// LS Electric XG5000 project: 과년68_3_3
// PLC NewPLC
// module base 0 slot 0: 입출력 모듈:XBC-DR20S (DC 24V 입력 12점, 릴레이 출력 8점)

PROGRAM NewProgram (task: 스캔 프로그램)

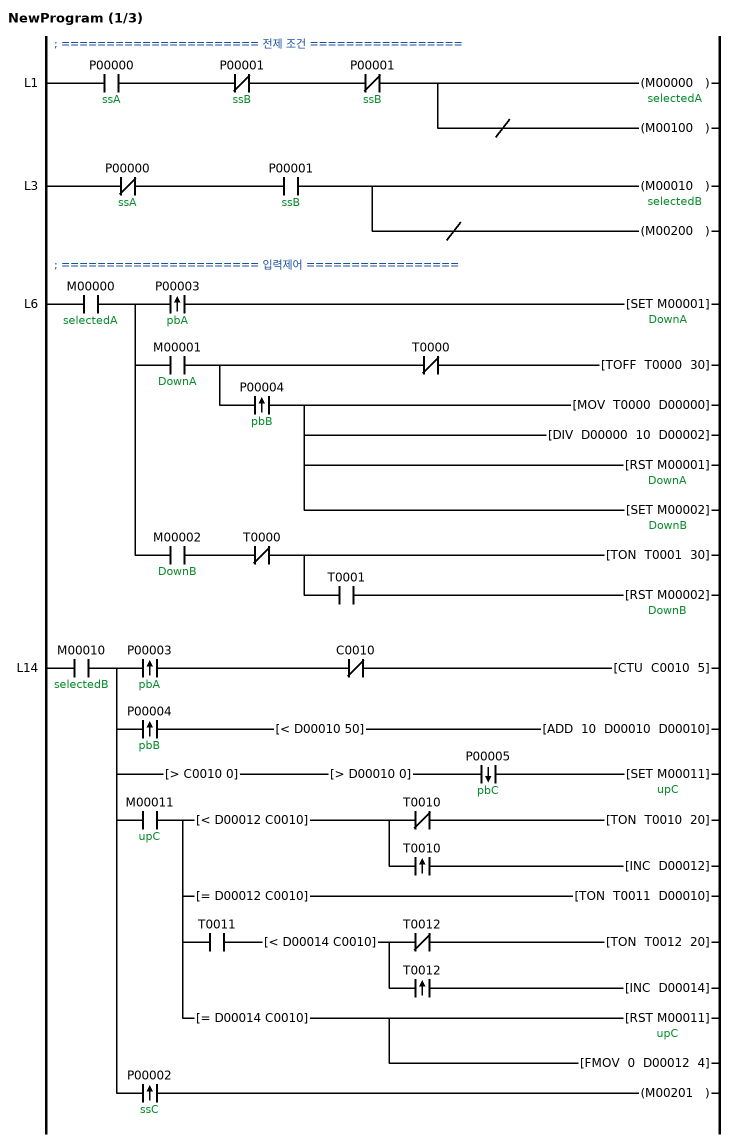
// ====================== 전제 조건 =================
; L1
LOAD      P00000	// ssA
AND NOT   P00001	// ssB
AND NOT   P00001	// ssB
OUT       M00000	// selectedA
NOT
OUT       M00100
; L3
LOAD NOT  P00000	// ssA
AND       P00001	// ssB
OUT       M00010	// selectedB
NOT
OUT       M00200
// ====================== 입력제어 =================
; L6
LOAD      M00000	// selectedA
MPUSH
ANDP      P00003	// pbA
SET       M00001	// DownA
MLOAD
AND       M00001	// DownA
MPUSH
AND NOT   T0000
TOFF      T0000 30
MPOP
ANDP      P00004	// pbB
MOV       T0000 D00000
DIV       D00000 10 D00002
RST       M00001	// DownA
SET       M00002	// DownB
MPOP
AND       M00002	// DownB
AND NOT   T0000
TON       T0001 30
AND       T0001
RST       M00002	// DownB
; L14
LOAD      M00010	// selectedB
MPUSH
ANDP      P00003	// pbA
AND NOT   C0010
CTU       C0010 5
MLOAD
ANDP      P00004	// pbB
AND<      D00010 50
ADD       10 D00010 D00010
MLOAD
AND>      C0010 0
AND>      D00010 0
ANDN      P00005	// pbC
SET       M00011	// upC
MLOAD
AND       M00011	// upC
MPUSH
AND<      D00012 C0010
MPUSH
AND NOT   T0010
TON       T0010 20
MPOP
ANDP      T0010
INC       D00012
MLOAD
AND=      D00012 C0010
TON       T0011 D00010
MLOAD
AND       T0011
AND<      D00014 C0010
MPUSH
AND NOT   T0012
TON       T0012 20
MPOP
ANDP      T0012
INC       D00014
MPOP
AND=      D00014 C0010
RST       M00011	// upC
FMOV      0 D00012 4
MPOP
ANDP      P00002	// ssC
OUT       M00201

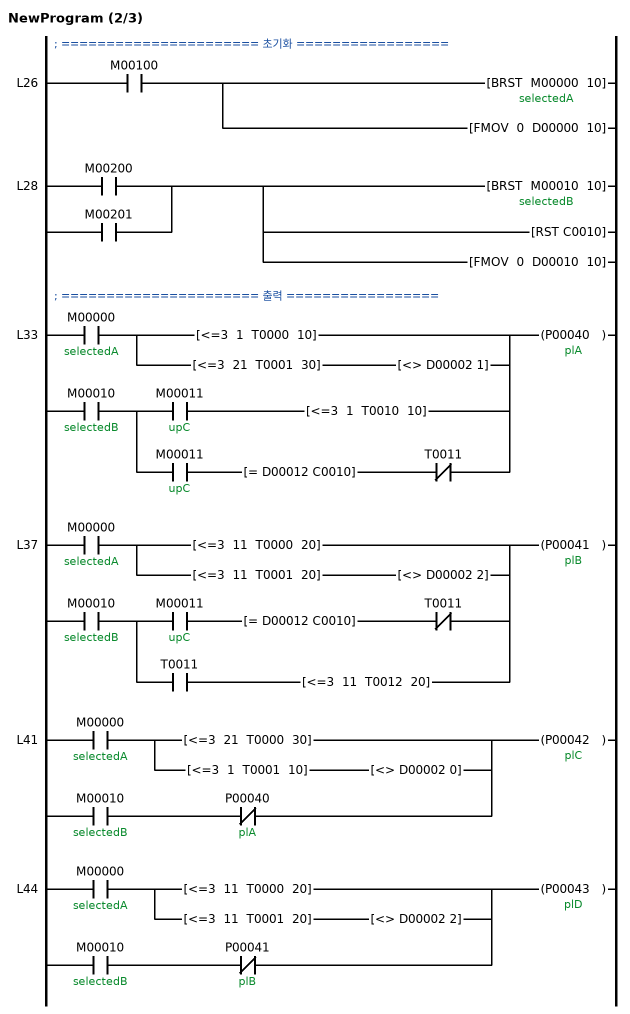
// ====================== 초기화 =================
; L26
LOAD      M00100
BRST      M00000 10	// selectedA
FMOV      0 D00000 10
; L28
LOAD      M00200
OR        M00201
BRST      M00010 10	// selectedB
RST       C0010
FMOV      0 D00010 10
// ====================== 출력 =================
; L33
LOAD      M00000	// selectedA
LOAD<=3   1 T0000 10
LOAD<=3   21 T0001 30
AND<>     D00002 1
OR LOAD
AND LOAD
LOAD      M00010	// selectedB
LOAD      M00011	// upC
AND<=3    1 T0010 10
LOAD      M00011	// upC
AND=      D00012 C0010
AND NOT   T0011
OR LOAD
AND LOAD
OR LOAD
OUT       P00040	// plA
; L37
LOAD      M00000	// selectedA
LOAD<=3   11 T0000 20
LOAD<=3   11 T0001 20
AND<>     D00002 2
OR LOAD
AND LOAD
LOAD      M00010	// selectedB
LOAD      M00011	// upC
AND=      D00012 C0010
AND NOT   T0011
LOAD      T0011
AND<=3    11 T0012 20
OR LOAD
AND LOAD
OR LOAD
OUT       P00041	// plB
; L41
LOAD      M00000	// selectedA
LOAD<=3   21 T0000 30
LOAD<=3   1 T0001 10
AND<>     D00002 0
OR LOAD
AND LOAD
LOAD      M00010	// selectedB
AND NOT   P00040	// plA
OR LOAD
OUT       P00042	// plC
; L44
LOAD      M00000	// selectedA
LOAD<=3   11 T0000 20
LOAD<=3   11 T0001 20
AND<>     D00002 2
OR LOAD
AND LOAD
LOAD      M00010	// selectedB
AND NOT   P00041	// plB
OR LOAD
OUT       P00043	// plD

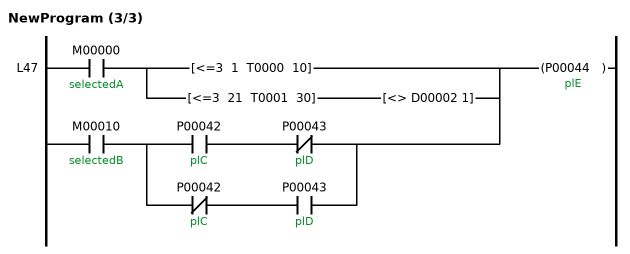
; L47
LOAD      M00000	// selectedA
LOAD<=3   1 T0000 10
LOAD<=3   21 T0001 30
AND<>     D00002 1
OR LOAD
AND LOAD
LOAD      M00010	// selectedB
LOAD      P00042	// plC
AND NOT   P00043	// plD
LOAD NOT  P00042	// plC
AND       P00043	// plD
OR LOAD
AND LOAD
OR LOAD
OUT       P00044	// plE